DATA_BLOCK "MEStoPLC"
{ S7_Optimized_Access := 'FALSE' }
VERSION : 0.1
NON_RETAIN
   STRUCT
      "MES.Load_Station1PartOK" : Bool;
      "MES.Load_Station1PartNG" : Bool;
      "MES.Load_Station1ReqMesDone" : Bool;
      Spare_1 : Bool;
      "MES.Load_Station2PartOK" : Bool;
      "MES.Load_Station2PartNG" : Bool;
      "MES.Load_Station2ReqMesDone" : Bool;
      Spare_2 : Bool;
      "MES.Load_Station3PartOK" : Bool;
      "MES.Load_Station3PartNG" : Bool;
      "MES.Load_Station3ReqMesDone" : Bool;
      Spare_3 : Bool;
      "MES.Load_Station4PartOK" : Bool;
      "MES.Load_Station4PartNG" : Bool;
      "MES.Load_Station4ReqMesDone" : Bool;
      Spare_4 : Bool;
      "MES.Load_Station5PartOK" : Bool;
      "MES.Load_Station5PartNG" : Bool;
      "MES.Load_Station5ReqMesDone" : Bool;
      Spare_5 : Bool;
      "MES.Load_Station6PartOK" : Bool;
      "MES.Load_Station6PartNG" : Bool;
      "MES.Load_Station6ReqMesDone" : Bool;
      Spare_6 : Bool;
      "MES.Load_Station7PartOK" : Bool;
      "MES.Load_Station7PartNG" : Bool;
      "MES.Load_Station7ReqMesDone" : Bool;
      Spare_7 : Bool;
      "MES.Load_Station8PartOK" : Bool;
      "MES.Load_Station8PartNG" : Bool;
      "MES.Load_Station8ReqMesDone" : Bool;
      Spare_8 : Bool;
      Spare_9 : Bool;
      Static_3 : Bool;
      "MES.Load_SubPart1OK" : Bool;
      "MES.Load_SubPart1tNG" : Bool;
      "MES.Load_SubPart1ReqMesDone" : Bool;
      Spare_10 : Bool;
      "MES.Load_SubPart2OK" : Bool;
      "MES.Load_SubPart2tNG" : Bool;
      "MES.Load_SubPart2ReqMesDone" : Bool;
      Spare_11 : Bool;
      "MES.Load_SubPart3OK" : Bool;
      "MES.Load_SubPart3tNG" : Bool;
      "MES.Load_SubPart3ReqMesDone" : Bool;
      Spare_12 : Bool;
      "MES.Load_SubPart4OK" : Bool;
      "MES.Load_SubPart4tNG" : Bool;
      "MES.Load_SubPart4ReqMesDone" : Bool;
      Spare_13 : Bool;
      "MES.Load_SubPart5OK" : Bool;
      "MES.Load_SubPart5tNG" : Bool;
      "MES.Load_SubPart5ReqMesDone" : Bool;
      Spare_14 : Bool;
      "MES.Load_SubPart6OK" : Bool;
      "MES.Load_SubPart6tNG" : Bool;
      "MES.Load_SubPart6ReqMesDone" : Bool;
      Spare_15 : Bool;
      "MES.Load_SubPart7OK" : Bool;
      "MES.Load_SubPart7tNG" : Bool;
      "MES.Load_SubPart7ReqMesDone" : Bool;
      Spare_16 : Bool;
      "MES.Load_SubPart8OK" : Bool;
      "MES.Load_SubPart8tNG" : Bool;
      "MES.Load_SubPart8ReqMesDone" : Bool;
      Spare : Bool;
      Spare_17 : Bool;
      "MES.Load_ResultsStored1OK" : Bool;
      "MES.Load_ResultsStored1NG" : Bool;
      "MES.Load_ResultsStored1ReqMesDone" : Bool;
      Spare_18 : Bool;
      "MES.Load_ResultsStored2OK" : Bool;
      "MES.Load_ResultsStored2NG" : Bool;
      "MES.Load_ResultsStored2ReqMesDone" : Bool;
      Spare_19 : Bool;
      "MES.Load_ResultsStored3OK" : Bool;
      "MES.Load_ResultsStored3NG" : Bool;
      "MES.Load_ResultsStored3ReqMesDone" : Bool;
      Spare_20 : Bool;
      "MES.Load_ResultsStored4OK" : Bool;
      "MES.Load_ResultsStored4NG" : Bool;
      "MES.Load_ResultsStored4ReqMesDone" : Bool;
      Spare_21 : Bool;
      "MES.Load_ResultsStored5OK" : Bool;
      "MES.Load_ResultsStored5NG" : Bool;
      "MES.Load_ResultsStored5ReqMesDone" : Bool;
      Spare_22 : Bool;
      "MES.Load_ResultsStored6OK" : Bool;
      "MES.Load_ResultsStored6NG" : Bool;
      "MES.Load_ResultsStored6ReqMesDone" : Bool;
      Spare_23 : Bool;
      "MES.Load_ResultsStored7OK" : Bool;
      "MES.Load_ResultsStored7NG" : Bool;
      "MES.Load_ResultsStored7ReqMesDone" : Bool;
      Spare_24 : Bool;
      "MES.Load_ResultsStored8OK" : Bool;
      "MES.Load_ResultsStored8NG" : Bool;
      "MES.Load_ResultsStored8ReqMesDone" : Bool;
      "MES.Load_StoveCheckInOk" : Bool;
      Static_1 : Bool;
      Spare_26 : Bool;
      Spare_27 : Bool;
      Spare_28 : Bool;
      Spare_29 : Bool;
      Spare_30 : Bool;
      Spare_31 : Bool;
      Spare_32 : Bool;
      Spare_33 : Bool;
      "MES.Unload_ResultsStored1OK" : Bool;
      "MES.Unload_ResultsStored1NG" : Bool;
      "MES.Unload_ResultsStored1ReqMesDone" : Bool;
      Spare_34 : Bool;
      "MES.Unload_ResultsStored2OK" : Bool;
      "MES.Unload_ResultsStored2NG" : Bool;
      "MES.Unload_ResultsStored2ReqMesDone" : Bool;
      Spare_35 : Bool;
      "MES.Unload_ResultsStored3OK" : Bool;
      "MES.Unload_ResultsStored3NG" : Bool;
      "MES.Unload_ResultsStored3ReqMesDone" : Bool;
      Spare_36 : Bool;
      "MES.Unload_ResultsStored4OK" : Bool;
      "MES.Unload_ResultsStored4NG" : Bool;
      "MES.Unload_ResultsStored4ReqMesDone" : Bool;
      Spare_37 : Bool;
      "MES.Unload_ResultsStored5OK" : Bool;
      "MES.Unload_ResultsStored5NG" : Bool;
      "MES.Unload_ResultsStored5ReqMesDone" : Bool;
      Spare_38 : Bool;
      "MES.Unload_ResultsStored6OK" : Bool;
      "MES.Unload_ResultsStored6NG" : Bool;
      "MES.Unload_ResultsStored6ReqMesDone" : Bool;
      Spare_39 : Bool;
      "MES.Unload_ResultsStored7OK" : Bool;
      "MES.Unload_ResultsStored7NG" : Bool;
      "MES.Unload_ResultsStored7ReqMesDone" : Bool;
      Spare_40 : Bool;
      "MES.Unload_ResultsStored8OK" : Bool;
      "MES.Unload_ResultsStored8NG" : Bool;
      "MES.Unload_ResultsStored8ReqMesDone" : Bool;
      Spare_41 : Bool;
      "MES.HeartbeatSignal" : Bool;
   END_STRUCT;


BEGIN

END_DATA_BLOCK

